// TIA Portal V19 export
TYPE "IPC_Msg_Log_MES"
   STRUCT
      Id : DInt;   // Identificativo progressivo univoco del messaggio (0 = cella vuota)
      timestamp : String;   // Timestamp evento formato ISO: YYYY-MM-DD HH:MM:SS.mmm
      topic : UDInt;   // Categoria/argomento del log per filtering e routing
      payLoad_1 : String;   // Descrizione del successo / insuccesso nell invio / ricezione
      payLoad_2 : String;   // Copia del messaggio inviato a MES / ricevuto da MES
   END_STRUCT;
END_TYPE
